// TwinCAT 3 PLC project MAS418_PLC
// ProgramVersion: 3.1.4023.0
// libraries:
//   Tc2_Standard, * (Beckhoff Automation GmbH)
//   Tc2_System, * (Beckhoff Automation GmbH)
//   Tc3_Module, * (Beckhoff Automation GmbH)
// project tree:
//   / PlcTask.TcTTO
//   POUs/ MAIN.TcPOU
//   Task1/ GVL_Task1.TcGVL, P_Task1.TcPOU

CONFIGURATION MAS418_PLC
    RESOURCE PLC ON TwinCAT3
        TASK PlcTask(INTERVAL := T#10ms, PRIORITY := 20);
        PROGRAM MAIN WITH PlcTask : MAIN;
    END_RESOURCE
END_CONFIGURATION

// ---- Task1/GVL_Task1.TcGVL
{attribute 'qualified_only'}
VAR_GLOBAL
	dtCurrentDt : DATE_AND_TIME := DT#2023-02-14-15:24:00;
	tVariable : TIME := T#5S;
END_VAR

// ---- POUs/MAIN.TcPOU
PROGRAM MAIN
VAR
END_VAR

P_Task1();

END_PROGRAM

// ---- Task1/P_Task1.TcPOU
PROGRAM P_Task1
VAR
	pPointer : POINTER TO DATE_AND_TIME := ADR(GVL_Task1.dtCurrentDt);
	tReference  : REFERENCE TO TIME REF=GVL_Task1.tVariable;
END_VAR

pPointer^ := DT#2023-02-08-15:31:19;
tReference := T#7S;

END_PROGRAM
